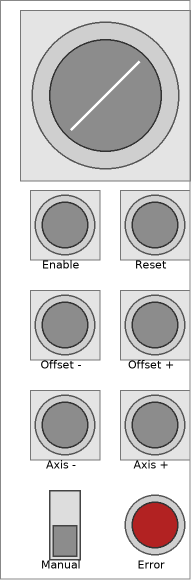
VISUALIZATION Pendant  // 191x580
    Potentiometer360 (20,10 171x171), style: Potentiometer-Potentiometer360-Gray, scale format: %.0f, scale 1..15
        p2431819421: Outside
    PushSwitch (30,190 70x70), behaviour: TOGGLE, style: Switch-PushSwitch-Gray
    Label (30,250 62x30), "Enable"
    PushSwitch (120,190 70x70), behaviour: TOGGLE, style: Switch-PushSwitch-Gray
    Label (120,250 62x30), "Reset"
    PushSwitch (30,290 70x70), behaviour: TOGGLE, style: Switch-PushSwitch-Gray
    Label (30,350 62x30), "Offset -"
    PushSwitch (120,290 70x70), behaviour: TOGGLE, style: Switch-PushSwitch-Gray
    Label (120,350 62x30), "Offset +"
    PushSwitch (30,390 70x70), behaviour: TOGGLE, style: Switch-PushSwitch-Gray
    Label (30,450 62x30), "Axis -"
    PushSwitch (120,390 70x70), behaviour: TOGGLE, style: Switch-PushSwitch-Gray
    Label (120,450 62x30), "Axis +"
    DipSwitch (30,490 70x70), behaviour: TOGGLE, style: Switch-DipSwitch-Gray
    Lamp1 (120,490 70x70), style: Lamp-Lamp1-Red
    Label (30,550 62x30), "Manual"
    Label (120,550 62x30), "Error"
END_VISUALIZATION

(* stored: Version 1.1.0.1, ProductVersion 3.1.4026.8
   Visu Pendant: Id {ccc5429d-fd15-4b7a-9efe-a44c0e8de7e0} *)
